// Mitsubishi GX Works2 project: Melsec   PLC: FX3U/FX3UC

PROGRAM MAIN
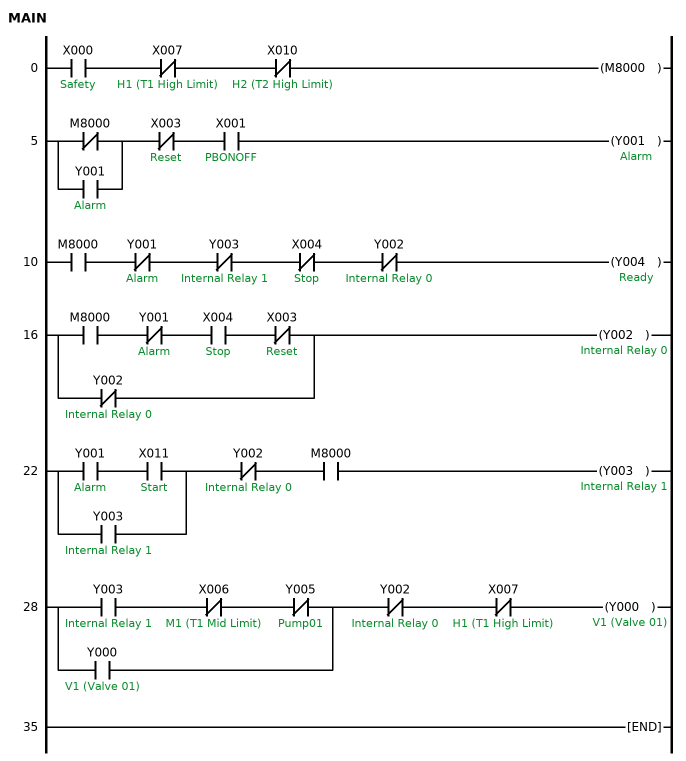
0     LD      X000  ; Safety
      ANI     X007  ; H1 (T1 High Limit)
      ANI     X010  ; H2 (T2 High Limit)
      OUT     M8000
5     LDI     M8000
      OR      Y001  ; Alarm
      ANI     X003  ; Reset
      AND     X001  ; PBONOFF
      OUT     Y001  ; Alarm
10    LD      M8000
      ANI     Y001  ; Alarm
      ANI     Y003  ; Internal Relay 1
      ANI     X004  ; Stop
      ANI     Y002  ; Internal Relay 0
      OUT     Y004  ; Ready
16    LD      M8000
      ANI     Y001  ; Alarm
      AND     X004  ; Stop
      ANI     X003  ; Reset
      ORI     Y002  ; Internal Relay 0
      OUT     Y002  ; Internal Relay 0
22    LD      Y001  ; Alarm
      AND     X011  ; Start
      OR      Y003  ; Internal Relay 1
      ANI     Y002  ; Internal Relay 0
      AND     M8000
      OUT     Y003  ; Internal Relay 1
28    LD      Y003  ; Internal Relay 1
      ANI     X006  ; M1 (T1 Mid Limit)
      ANI     Y005  ; Pump01
      OR      Y000  ; V1 (Valve 01)
      ANI     Y002  ; Internal Relay 0
      ANI     X007  ; H1 (T1 High Limit)
      OUT     Y000  ; V1 (Valve 01)
35    END
END_PROGRAM

// device comments not shown above
X002  ; PBEstop
X005  ; L1 (T1 Low Limit)
M4000  ; Internal Safety Relay
